{attribute 'qualified_only'}
VAR_GLOBAL
	g_fbMenu :  FB_VisuMenu;
END_VAR

(* stored: Version 1.1.0.1, ProductVersion 3.1.4026.13
   GVL GVL_Visu: Id {b83a4829-5a57-42e1-b02b-16db40162563} *)
